FUNCTION_BLOCK FB_AnalogSensor_full
VAR_INPUT
	lettura			:INT;
	maxScaleBit		:INT;
	maxScaleIng		:INT;
	deltaLowLimit	:INT;
	distanzaAVuoto	:INT;
	valSoglia		:INT;
	filterTime		:INT;		//seconds
END_VAR
VAR_OUTPUT
	full			:BOOL;
	actualVal		:INT;
END_VAR
VAR
	_actVal			:INT;
	_tmr			:TON;
	_over			:BOOL;
END_VAR


_actVal := ((lettura*maxScaleIng)/maxScaleBit) - deltaLowLimit;
actualVal:=_actVal ;
IF distanzaAVuoto - _actVal > valSoglia THEN
	_over := TRUE;
ELSE
	full:=FALSE;
END_IF

_tmr(IN:=_over, PT:=INT_TO_TIME(filterTime*1000));
IF _tmr.Q THEN
	_over:=FALSE;
	full:=TRUE;
END_IF

END_FUNCTION_BLOCK

(* stored: Version 1.1.0.1, ProductVersion 3.1.4022.12
   POU FB_AnalogSensor_full: Id {01cab774-f576-4878-a10f-dc30a7c8f7b3}, SpecialFunc None *)
